FUNCTION_BLOCK FB_Bridge_Inputs_Real
// Interface with 20 ports. Converts UDINT to REAL (32 bits)
VAR_INPUT
	I00 : UDINT := 0;	// Input real 00
	I01 : UDINT := 0;	// Input real 01
	I02 : UDINT := 0;	// Input real 02
	I03 : UDINT := 0;	// Input real 03
	I04 : UDINT := 0;	// Input real 04
	I05 : UDINT := 0;	// Input real 05
	I06 : UDINT := 0;	// Input real 06
	I07 : UDINT := 0;	// Input real 07
	I08 : UDINT := 0;	// Input real 08
	I09 : UDINT := 0;	// Input real 09
	I10 : UDINT := 0;	// Input real 10
	I11 : UDINT := 0;	// Input real 11
	I12 : UDINT := 0;	// Input real 12
	I13 : UDINT := 0;	// Input real 13
	I14 : UDINT := 0;	// Input real 14
	I15 : UDINT := 0;	// Input real 15
	I16 : UDINT := 0;	// Input real 16
	I17 : UDINT := 0;	// Input real 17
	I18 : UDINT := 0;	// Input real 18
	I19 : UDINT := 0;	// Input real 19
END_VAR
VAR_OUTPUT
	Q00 : REAL;
	Q01 : REAL;
	Q02 : REAL;
	Q03 : REAL;
	Q04 : REAL;
	Q05 : REAL;
	Q06 : REAL;
	Q07 : REAL;
	Q08 : REAL;
	Q09 : REAL;
	Q10 : REAL;
	Q11 : REAL;
	Q12 : REAL;
	Q13 : REAL;
	Q14 : REAL;
	Q15 : REAL;
	Q16 : REAL;
	Q17 : REAL;
	Q18 : REAL;
	Q19 : REAL;
END_VAR
VAR
END_VAR

Q00 := DW_TO_REAL(I00);
Q01 := DW_TO_REAL(I01);
Q02 := DW_TO_REAL(I02);
Q03 := DW_TO_REAL(I03);
Q04 := DW_TO_REAL(I04);
Q05 := DW_TO_REAL(I05);
Q06 := DW_TO_REAL(I06);
Q07 := DW_TO_REAL(I07);
Q08 := DW_TO_REAL(I08);
Q09 := DW_TO_REAL(I09);
Q10 := DW_TO_REAL(I10);
Q11 := DW_TO_REAL(I11);
Q12 := DW_TO_REAL(I12);
Q13 := DW_TO_REAL(I13);
Q14 := DW_TO_REAL(I14);
Q15 := DW_TO_REAL(I15);
Q16 := DW_TO_REAL(I16);
Q17 := DW_TO_REAL(I17);
Q18 := DW_TO_REAL(I18);
Q19 := DW_TO_REAL(I19);

END_FUNCTION_BLOCK

(* stored: Version 1.1.0.1, ProductVersion 3.1.4024.9
   POU FB_Bridge_Inputs_Real: Id {1100369f-d7fa-446a-962a-a8af348a2ffe}, SpecialFunc None *)
